CASE nStep OF
    0:
        // Set the thermocouple temperatures to crazy high number
        SetPPMTemp(100);
        nStep := nStep + 1;
    1:
        // Wait till we see "OUT" state and one other state (OUT should be no fault)
        IF fbPPM.eEnumGet = E_PPM_States.OUT THEN
            AssertNeitherTempFault('was in out position');
            bOutChecked := TRUE;
        ELSIF fbPPM.eEnumGet <> E_PPM_States.Unknown THEN
            AssertBothTempFault('was in a target position');
            bInChecked := TRUE;
        END_IF
        IF bOutChecked AND bInChecked THEN
            nStep := nStep + 1;
        END_IF
    2:
        // Set the thermocouple temperatures to low again
        SetPPMTemp(0);
        nStep := nStep + 1;
    3:
        AssertNeitherTempFault('has low temp reading');
        nStep := nStep + 1;
END_CASE;

IF tonTimer.Q OR nStep > nLastStep THEN
    AssertFalse(tonTimer.Q, 'Timeout in PPM temp FFO test');
    TEST_FINISHED();
END_IF
END_METHOD

END_FUNCTION_BLOCK

// Tests/FB_REFTest
FUNCTION_BLOCK FB_REFTest EXTENDS FB_TestSuite
VAR
    fbREF: FB_REF;
    stYStage: ST_MotionStage;

    stDefault: ST_PositionState := (
        fVelocity:=10,
        bMoveOk:=TRUE,
        bValid:=TRUE
    );
    fbSetup: FB_StateSetupHelper;

    fbFFHWO: FB_HardwareFFOutput;
    fbArbiter: FB_Arbiter(1);
    fbSubSysIO: FB_DummyArbIO;

    bInit: BOOL;
END_VAR

// Fake PMPS handling
fbSubSysIO(
    LA:=fbArbiter,
    FFO:=fbFFHWO,
);

// Fake limit handling
stYStage.bLimitBackwardEnable := TRUE;
stYStage.bLimitForwardEnable := TRUE;

// Standard state setup
fbSetup(stPositionState:=stDefault, bSetDefault:=TRUE);
fbSetup(stPositionState:=fbREF.stOut, sName:='OUT', fPosition:=10, sPmpsState:='T0');
fbSetup(stPositionState:=fbREF.stIn, sName:='T1', fPosition:=20, sPmpsState:='T1');

// Standard FB call
fbREF(
    stYStage:=stYStage,
    fbFFHWO:=fbFFHWO,
    fbArbiter:=fbArbiter,
    bEnableMotion:=TRUE,
    bEnableBeamParams:=TRUE,
    bEnablePositionLimits:=TRUE,
    sDeviceName:='DEVICE',
    sTransitionKey:='T9',
    bReadDBNow:=NOT bInit,
);

TestStateMove();

bInit := TRUE;

METHOD TestStateMove
VAR_INST
    tonTimer: TON;
    nIterState: UINT := 0;
END_VAR
VAR CONSTANT
    nLastState: UINT := E_EpicsInOut.IN;
END_VAR

// Sanity check: can we at least move to every named state?
TEST('TestREFStateMove');

// Prepare a timeout
tonTimer(IN:=TRUE, PT:=T#10s);

// Start in Unknown, then go through the state positions one by one
IF fbREF.eEnumGet = nIterState THEN
    nIterState := nIterState + 1;
    fbREF.eEnumSet := nIterState;
END_IF

IF tonTimer.Q OR nIterState > nLastState THEN
    AssertFalse(tonTimer.Q, 'Timeout in REF move test');
    TEST_FINISHED();
END_IF
END_METHOD

END_FUNCTION_BLOCK

// Tests/FB_SATTTest
FUNCTION_BLOCK FB_SATTTest EXTENDS FB_TestSuite
VAR
    fbSATT: FB_SXR_SATT_Stage;
    stYStage: ST_MotionStage;

    stDefault: ST_PositionState := (
        fDelta:=0.5,
        fVelocity:=10,
        bMoveOk:=TRUE,
        bValid:=TRUE
    );
    fbSetup: FB_StateSetupHelper;

    fbFFHWO: FB_HardwareFFOutput;

    bInit: BOOL;
END_VAR

// Fake limit handling
stYStage.bLimitBackwardEnable := TRUE;
stYStage.bLimitForwardEnable := TRUE;

// Standard state setup
fbSetup(stPositionState:=stDefault, bSetDefault:=TRUE);
fbSetup(stPositionState:=fbSATT.stOut, sName:='OUT', fPosition:=10);
fbSetup(stPositionState:=fbSATT.stFilter1, sName:='T1', fPosition:=20, sPmpsState:='T1');
fbSetup(stPositionState:=fbSATT.stFilter2, sName:='T2', fPosition:=30);
fbSetup(stPositionState:=fbSATT.stFilter3, sName:='T3', fPosition:=40);
fbSetup(stPositionState:=fbSATT.stFilter4, sName:='T4', fPosition:=50);
fbSetup(stPositionState:=fbSATT.stFilter5, sName:='T5', fPosition:=60);
fbSetup(stPositionState:=fbSATT.stFilter6, sName:='T6', fPosition:=70);
fbSetup(stPositionState:=fbSATT.stFilter7, sName:='T7', fPosition:=80);
fbSetup(stPositionState:=fbSATT.stFilter8, sName:='T8', fPosition:=90);

// Standard FB call
fbSATT(
    stAxis:=stYStage,
    fbFFHWO:=fbFFHWO,
    bEnable:=TRUE,
    sDeviceName:='DEVICE',
);

TestStateMove();
TestTempFFO();

bInit := TRUE;

METHOD AssertBothTempFault
VAR_INPUT
    Message: STRING;
END_VAR

AssertFalse(
    fbSATT.fbRTD_1.FFO.i_xOK,
    CONCAT('SATT RTD1 expected fault: ', Message),
);
AssertFalse(
    fbSATT.fbRTD_2.FFO.i_xOK,
    CONCAT('SATT RTD2 expected fault: ', Message),
);
END_METHOD

METHOD AssertNeitherTempFault
VAR_INPUT
    Message: STRING;
END_VAR

AssertTrue(
    fbSATT.fbRTD_1.FFO.i_xOK,
    CONCAT('SATT RTD1 expected ok: ', Message),
);
AssertTrue(
    fbSATT.fbRTD_2.FFO.i_xOK,
    CONCAT('SATT RTD2 expected ok: ', Message),
);
END_METHOD

METHOD SetSATTTemp
VAR_INPUT
    iTempC: INT;
END_VAR
VAR
    ptr: POINTER TO INT;
END_VAR

ptr := ADR(fbSATT.fbRTD_1.iRaw);
ptr^ := iTempC * 100;

ptr := ADR(fbSATT.fbRTD_2.iRaw);
ptr^ := iTempC * 100;
END_METHOD

METHOD TestStateMove
VAR_INST
    tonTimer: TON;
    nIterState: UINT := 0;
END_VAR
VAR CONSTANT
    nLastState: UINT := E_SXR_SATT_Position.FILTER8;
END_VAR

// Sanity check: can we at least move to every named state?
TEST('TestSATTStateMove');

// Prepare a timeout
tonTimer(IN:=TRUE, PT:=T#20s);

// Start in Unknown, then go through the state positions one by one
IF fbSATT.eEnumGet = nIterState THEN
    nIterState := nIterState + 1;
    fbSATT.eEnumSet := nIterState;
END_IF

IF tonTimer.Q OR nIterState > nLastState THEN
    AssertFalse(tonTimer.Q, 'Timeout in SATT move test');
    TEST_FINISHED();
END_IF
END_METHOD

METHOD TestTempFFO
VAR_INST
    tonTimer: TON;
    nStep: UINT := 0;
    bOutChecked: BOOL := FALSE;
    bInChecked: BOOL := FALSE;
END_VAR
VAR CONSTANT
    nLastStep: UINT := 3;
END_VAR

// Do we fault at the correct times?
// Parasitically depends on state move test
TEST('TestSATTTempFFO');

// Prepare a timeout
tonTimer(IN:=TRUE, PT:=T#10s);

CASE nStep OF
    0:
        // Set the thermocouple temperatures to crazy high number
        SetSATTTemp(100);
        nStep := nStep + 1;
    1:
        // Wait till we see "OUT" state and one other state (OUT should be no fault)
        IF fbSATT.eEnumGet = E_SXR_SATT_Position.OUT THEN
            AssertNeitherTempFault('was in out position');
            bOutChecked := TRUE;
        ELSIF fbSATT.eEnumGet <> E_SXR_SATT_Position.Unknown THEN
            AssertBothTempFault('was in a target position');
            bInChecked := TRUE;
        END_IF
        IF bOutChecked AND bInChecked THEN
            nStep := nStep + 1;
        END_IF
    2:
        // Set the thermocouple temperatures to low again
        SetSATTTemp(0);
        nStep := nStep + 1;
    3:
        AssertNeitherTempFault('has low temp reading');
        nStep := nStep + 1;
END_CASE;

IF tonTimer.Q OR nStep > nLastStep THEN
    AssertFalse(tonTimer.Q, 'Timeout in SATT temp FFO test');
    TEST_FINISHED();
END_IF
END_METHOD

END_FUNCTION_BLOCK

// Tests/FB_SLITS_POWERTest
FUNCTION_BLOCK FB_SLITS_POWERTest EXTENDS FB_TestSuite
VAR
    fbSlitsPower: FB_SLITS_POWER;
    M1: ST_MotionStage;
    M2: ST_MotionStage;
    M3: ST_MotionStage;
    M4: ST_MotionStage;
    bExecuteMotion: BOOL := FALSE;

    fbFFHWO: FB_HardwareFFOutput;
    fbArbiter: FB_Arbiter(1);
END_VAR

fbSlitsPower(
    stTopBlade:=M1,
    stBottomBlade:=M2,
    stNorthBlade:=M3,
    stSouthBlade:=M4,
    bExecuteMotion:=bExecuteMotion,
    i_DevName:='DEVICE',
    sPmpsState:='T1',
    io_fbFFHWO := fbFFHWO,
    fbArbiter := fbArbiter,
);

TestTempFFO();

METHOD AssertAllTempFault
VAR_INPUT
    Message: STRING;
END_VAR

AssertFalse(
    fbSlitsPower.RTD_TOP_1.FFO.i_xOK,
    CONCAT('Slits Top 1 RTD expected fault: ', Message),
);
AssertFalse(
    fbSlitsPower.RTD_TOP_2.FFO.i_xOK,
    CONCAT('Slits Top 2 RTD expected fault: ', Message),
);
AssertFalse(
    fbSlitsPower.RTD_Bottom_1.FFO.i_xOK,
    CONCAT('Slits Bottom 1 RTD expected fault: ', Message),
);
AssertFalse(
    fbSlitsPower.RTD_Bottom_2.FFO.i_xOK,
    CONCAT('Slits Bottom 2 RTD expected fault: ', Message),
);
AssertFalse(
    fbSlitsPower.RTD_North_1.FFO.i_xOK,
    CONCAT('Slits North 1 RTD expected fault: ', Message),
);
AssertFalse(
    fbSlitsPower.RTD_North_2.FFO.i_xOK,
    CONCAT('Slits North 2 RTD expected fault: ', Message),
);
AssertFalse(
    fbSlitsPower.RTD_South_1.FFO.i_xOK,
    CONCAT('Slits South 1 RTD expected fault: ', Message),
);
AssertFalse(
    fbSlitsPower.RTD_South_2.FFO.i_xOK,
    CONCAT('Slits South 2 1 RTD expected fault: ', Message),
);
END_METHOD

METHOD AssertNoneTempFault
VAR_INPUT
    Message: STRING;
END_VAR

AssertTrue(
    fbSlitsPower.RTD_TOP_1.FFO.i_xOK,
    CONCAT('Slits Top 1 RTD expected ok: ', Message),
);
AssertTrue(
    fbSlitsPower.RTD_TOP_2.FFO.i_xOK,
    CONCAT('Slits Top 2 RTD expected ok: ', Message),
);
AssertTrue(
    fbSlitsPower.RTD_Bottom_1.FFO.i_xOK,
    CONCAT('Slits Bottom 1 RTD expected ok: ', Message),
);
AssertTrue(
    fbSlitsPower.RTD_Bottom_2.FFO.i_xOK,
    CONCAT('Slits Bottom 2 RTD expected ok: ', Message),
);
AssertTrue(
    fbSlitsPower.RTD_North_1.FFO.i_xOK,
    CONCAT('Slits North 1 RTD expected ok: ', Message),
);
AssertTrue(
    fbSlitsPower.RTD_North_2.FFO.i_xOK,
    CONCAT('Slits North 2 RTD expected ok: ', Message),
);
AssertTrue(
    fbSlitsPower.RTD_South_1.FFO.i_xOK,
    CONCAT('Slits South 1 RTD expected ok: ', Message),
);
AssertTrue(
    fbSlitsPower.RTD_South_2.FFO.i_xOK,
    CONCAT('Slits South 2 1 RTD expected ok: ', Message),
);
END_METHOD

METHOD SetSlitsTemp
VAR_INPUT
    iTempC: INT;
END_VAR
VAR
    ptr: POINTER TO INT;
END_VAR

ptr := ADR(fbSlitsPower.RTD_TOP_1.iRaw);
ptr^ := iTempC * 10;

ptr := ADR(fbSlitsPower.RTD_TOP_2.iRaw);
ptr^ := iTempC * 10;

ptr := ADR(fbSlitsPower.RTD_Bottom_1.iRaw);
ptr^ := iTempC * 10;

ptr := ADR(fbSlitsPower.RTD_Bottom_2.iRaw);
ptr^ := iTempC * 10;

ptr := ADR(fbSlitsPower.RTD_North_1.iRaw);
ptr^ := iTempC * 10;

ptr := ADR(fbSlitsPower.RTD_North_2.iRaw);
ptr^ := iTempC * 10;

ptr := ADR(fbSlitsPower.RTD_South_1.iRaw);
ptr^ := iTempC * 10;

ptr := ADR(fbSlitsPower.RTD_South_2.iRaw);
ptr^ := iTempC * 10;
END_METHOD

METHOD TestTempFFO
VAR_INST
    tonTimer: TON;
    nStep: UINT := 0;
END_VAR
VAR CONSTANT
    nLastStep: UINT := 4;
END_VAR

// Do we fault at the correct times?
TEST('TestSlitsTempFFO');

// Prepare a timeout
tonTimer(IN:=TRUE, PT:=T#10s);


CASE nStep OF
    0:
        // Hold until the PMPS DB is ready
        // Most tests don't need this because they start by waiting for a move
        IF fbSlitsPower.RTD_TOP_1.fFaultThreshold > 0 THEN
            nStep := nStep + 1;
        END_IF
    1:
        // Set the thermocouple temperatures to crazy high number
        SetSlitsTemp(100);
        nStep := nStep + 1;
    2:
        // We should see faults on all RTDs at 100C
        AssertAllTempFault('has high temp reading');
        nStep := nStep + 1;
    3:
        // Set the thermocouple temperatures to low again
        SetSlitsTemp(0);
        nStep := nStep + 1;
    4:
        AssertNoneTempFault('has low temp reading');
        nStep := nStep + 1;
END_CASE;

IF tonTimer.Q OR nStep > nLastStep THEN
    AssertFalse(tonTimer.Q, 'Timeout in PPM temp FFO test');
    TEST_FINISHED();
END_IF
END_METHOD

END_FUNCTION_BLOCK

// Tests/FB_WFSTest
FUNCTION_BLOCK FB_WFSTest EXTENDS FB_TestSuite
VAR
    fbWFS: FB_WFS;
    stYStage: ST_MotionStage;
    stZStage: ST_MotionStage;

    stDefault: ST_PositionState := (
        fVelocity:=10,
        bMoveOk:=TRUE,
        bValid:=TRUE
    );
    fbSetup: FB_StateSetupHelper;

    fbFFHWO: FB_HardwareFFOutput;
    fbArbiter: FB_Arbiter(1);
    fbSubSysIO: FB_DummyArbIO;

    bInit: BOOL;
END_VAR

// Fake PMPS handling
fbSubSysIO(
    LA:=fbArbiter,
    FFO:=fbFFHWO,
);

// Fake limit handling
stYStage.bLimitBackwardEnable := TRUE;
stYStage.bLimitForwardEnable := TRUE;

// Standard state setup
fbSetup(stPositionState:=stDefault, bSetDefault:=TRUE);
fbSetup(stPositionState:=fbWFS.stOut, sName:='OUT', fPosition:=10, sPmpsState:='T0');
fbSetup(stPositionState:=fbWFS.stTarget1, sName:='T1', fPosition:=20, sPmpsState:='T1');
fbSetup(stPositionState:=fbWFS.stTarget2, sName:='T2', fPosition:=30, sPmpsState:='T2');
fbSetup(stPositionState:=fbWFS.stTarget3, sName:='T3', fPosition:=40, sPmpsState:='T3');
fbSetup(stPositionState:=fbWFS.stTarget4, sName:='T4', fPosition:=50, sPmpsState:='T4');
fbSetup(stPositionState:=fbWFS.stTarget5, sName:='T5', fPosition:=60, sPmpsState:='T5');

// Standard FB call
fbWFS(
    stYStage:=stYStage,
    stZStage:=stZStage,
    fbFFHWO:=fbFFHWO,
    fbArbiter:=fbArbiter,
    bEnableMotion:=TRUE,
    bEnableBeamParams:=TRUE,
    bEnablePositionLimits:=TRUE,
    sDeviceName:='DEVICE',
    sTransitionKey:='T9',
    bReadDBNow:=NOT bInit,
);

TestStateMove();
TestTempFFO();

bInit := TRUE;

METHOD AssertBothTempFault
VAR_INPUT
    Message: STRING;
END_VAR

AssertFalse(
    fbWFS.fbThermoCouple1.FFO.i_xOK,
    CONCAT('WFS TC1 expected fault: ', Message),
);
AssertFalse(
    fbWFS.fbThermoCouple2.FFO.i_xOK,
    CONCAT('WFS TC2 expected fault: ', Message),
);
END_METHOD

METHOD AssertNeitherTempFault
VAR_INPUT
    Message: STRING;
END_VAR

AssertTrue(
    fbWFS.fbThermoCouple1.FFO.i_xOK,
    CONCAT('WFS TC1 expected ok: ', Message),
);
AssertTrue(
    fbWFS.fbThermoCouple1.FFO.i_xOK,
    CONCAT('WFS TC2 sensor expected ok: ', Message),
);
END_METHOD

METHOD SetWFSTemp
VAR_INPUT
    iTempC: INT;
END_VAR
VAR
    ptr: POINTER TO INT;
END_VAR

ptr := ADR(fbWFS.fbThermoCouple1.iRaw);
ptr^ := iTempC * 10;

ptr := ADR(fbWFS.fbThermoCouple2.iRaw);
ptr^ := iTempC * 10;
END_METHOD

METHOD TestStateMove
VAR_INST
    tonTimer: TON;
    nIterState: UINT := 0;
END_VAR
VAR CONSTANT
    nLastState: UINT := E_WFS_States.TARGET5;
END_VAR

// Sanity check: can we at least move to every named state?
TEST('TestWFSStateMove');

// Prepare a timeout
tonTimer(IN:=TRUE, PT:=T#10s);

// Start in Unknown, then go through the state positions one by one
IF fbWFS.eEnumGet = nIterState THEN
    nIterState := nIterState + 1;
    fbWFS.eEnumSet := nIterState;
END_IF

IF tonTimer.Q OR nIterState > nLastState THEN
    AssertFalse(tonTimer.Q, 'Timeout in WFS move test');
    TEST_FINISHED();
END_IF
END_METHOD

METHOD TestTempFFO
VAR_INST
    tonTimer: TON;
    nStep: UINT := 0;
    bOutChecked: BOOL := FALSE;
    bInChecked: BOOL := FALSE;
END_VAR
VAR CONSTANT
    nLastStep: UINT := 3;
END_VAR

// Do we fault at the correct times?
// Parasitically depends on state move test
TEST('TestWFSTempFFO');

// Prepare a timeout
tonTimer(IN:=TRUE, PT:=T#10s);

CASE nStep OF
    0:
        // Set the thermocouple temperatures to crazy high number
        SetWFSTemp(100);
        nStep := nStep + 1;
    1:
        // Wait till we see "OUT" state and one other state (OUT should be no fault)
        IF fbWFS.eEnumGet = E_WFS_States.OUT THEN
            AssertNeitherTempFault('was in out position');
            bOutChecked := TRUE;
        ELSIF fbWFS.eEnumGet <> E_WFS_States.Unknown THEN
            AssertBothTempFault('was in a target position');
            bInChecked := TRUE;
        END_IF
        IF bOutChecked AND bInChecked THEN
            nStep := nStep + 1;
        END_IF
    2:
        // Set the thermocouple temperatures to low again
        SetWFSTemp(0);
        nStep := nStep + 1;
    3:
        AssertNeitherTempFault('has low temp reading');
        nStep := nStep + 1;
END_CASE;

IF tonTimer.Q OR nStep > nLastStep THEN
    AssertFalse(tonTimer.Q, 'Timeout in WFS temp FFO test');
    TEST_FINISHED();
END_IF
END_METHOD

END_FUNCTION_BLOCK

// Tests/FB_XPIMTest
FUNCTION_BLOCK FB_XPIMTest EXTENDS FB_TestSuite
VAR
    fbXPIM: FB_XPIM;
    stYStage: ST_MotionStage;
    stZoomStage: ST_MotionStage;
    stFocusStage: ST_MotionStage;

    stEl6In: EL6inData22b;
    stEl6Out: EL6OutData22b;

    stDefault: ST_PositionState := (
        fVelocity:=10,
        bMoveOk:=TRUE,
        bValid:=TRUE
    );
    fbSetup: FB_StateSetupHelper;

    fbFFHWO: FB_HardwareFFOutput;
    fbArbiter: FB_Arbiter(1);
    fbSubSysIO: FB_DummyArbIO;

    bInit: BOOL;
END_VAR

// Fake PMPS handling
fbSubSysIO(
    LA:=fbArbiter,
    FFO:=fbFFHWO,
);

// Fake limit handling
stYStage.bLimitBackwardEnable := TRUE;
stYStage.bLimitForwardEnable := TRUE;

// Standard state setup
fbSetup(stPositionState:=stDefault, bSetDefault:=TRUE);
fbSetup(stPositionState:=fbXPIM.stOut, sName:='OUT', fPosition:=10, sPmpsState:='T0');
fbSetup(stPositionState:=fbXPIM.stReticle, sName:='T1', fPosition:=20, sPmpsState:='T1');
fbSetup(stPositionState:=fbXPIM.stYag, sName:='T2', fPosition:=30, sPmpsState:='T2');
fbSetup(stPositionState:=fbXPIM.stDiamond, sName:='T3', fPosition:=40, sPmpsState:='T3');

// Standard FB call
fbXPIM(
    stYStage:=stYStage,
    stZoomStage:=stZoomStage,
    stFocusStage:=stFocusStage,
    fbFFHWO:=fbFFHWO,
    fbArbiter:=fbArbiter,
    stEl6In:=stEl6In,
    stEl6Out:=stEl6Out,
    bEnableMotion:=TRUE,
    bEnableBeamParams:=TRUE,
    bEnablePositionLimits:=TRUE,
    sDeviceName:='DEVICE',
    sTransitionKey:='T9',
    bReadDBNow:=NOT bInit,
);

TestStateMove();

bInit := TRUE;

METHOD TestStateMove
VAR_INST
    tonTimer: TON;
    nIterState: UINT := 0;
END_VAR
VAR CONSTANT
    nLastState: UINT := E_XPIM_States.RETICLE;
END_VAR

// Sanity check: can we at least move to every named state?
TEST('TestXPIMStateMove');

// Prepare a timeout
tonTimer(IN:=TRUE, PT:=T#10s);

// Start in Unknown, then go through the state positions one by one
IF fbXPIM.eEnumGet = nIterState THEN
    nIterState := nIterState + 1;
    fbXPIM.eEnumSet := nIterState;
END_IF

IF tonTimer.Q OR nIterState > nLastState THEN
    AssertFalse(tonTimer.Q, 'Timeout in XPIM move test');
    TEST_FINISHED();
END_IF
END_METHOD

END_FUNCTION_BLOCK

// Tests/PRG_TEST
{attribute 'analysis' := '-33'}
PROGRAM PRG_TEST
VAR
    fbATMTest: FB_ATMTest;
    fbLICTest: FB_LICTest;
    fbPPMTest: FB_PPMTest;
    fbREFTest: FB_REFTest;
    fbSATTTest: FB_SATTTest;
    fbSlitsPowerTest: FB_SLITS_POWERTest;
    fbWFSTest: FB_WFSTest;
    fbXPIMTest: FB_XPIMTest;
    fbCheckPositionStateWriteTest: FB_CheckPositionStateWriteTest;
    fbCCTempSensorTest: FB_CC_TempSensorTest;

    fbSetupJson: FB_PMPSJsonTestHelper;
    astBeamParams: ARRAY[0..9] OF ST_DbStateParams;
    nIter: UINT;
END_VAR


// Setup a fake db export for the test suite
FOR nIter := 0 TO 9 DO
    astBeamParams[nIter].stBeamParams := PMPS_GVL.cstFullBeam;
    astBeamParams[nIter].sPmpsState := CONCAT('T', UINT_TO_STRING(nIter));
    astBeamParams[nIter].stReactiveParams.nTempSP := nIter + 20;
END_FOR
fbSetupJson(
    astBeamParams := astBeamParams,
    bExecute := TRUE,
    sDevNAme := 'DEVICE',
);
// Run the tests
TcUnit.RUN();

END_PROGRAM
